// TIA Portal V20 export
FUNCTION "07 T5 EXCENTRIC LEV2" : Void   // FC1718, LAD
TITLE = TRACKING - LEV2
{ S7_Optimized_Access := 'TRUE' }
// stored: AutoNumber false, SetENOAutomatically false
   VAR_TEMP
      "HSK Answer OK" : Bool;
      Trc_OK : Bool;
      Aux_Int : Int;
      Aux_Bool : Bool;
   END_VAR
   VAR_TEMP   // added for the SCL form of the ladder/FBD networks
      _w1 : Bool;
      _w2 : Bool;
      _w3 : Bool;
   END_VAR
BEGIN

REGION Network 1: ============ Manual movement ============
END_REGION

REGION Network 2: pipe trasnfered
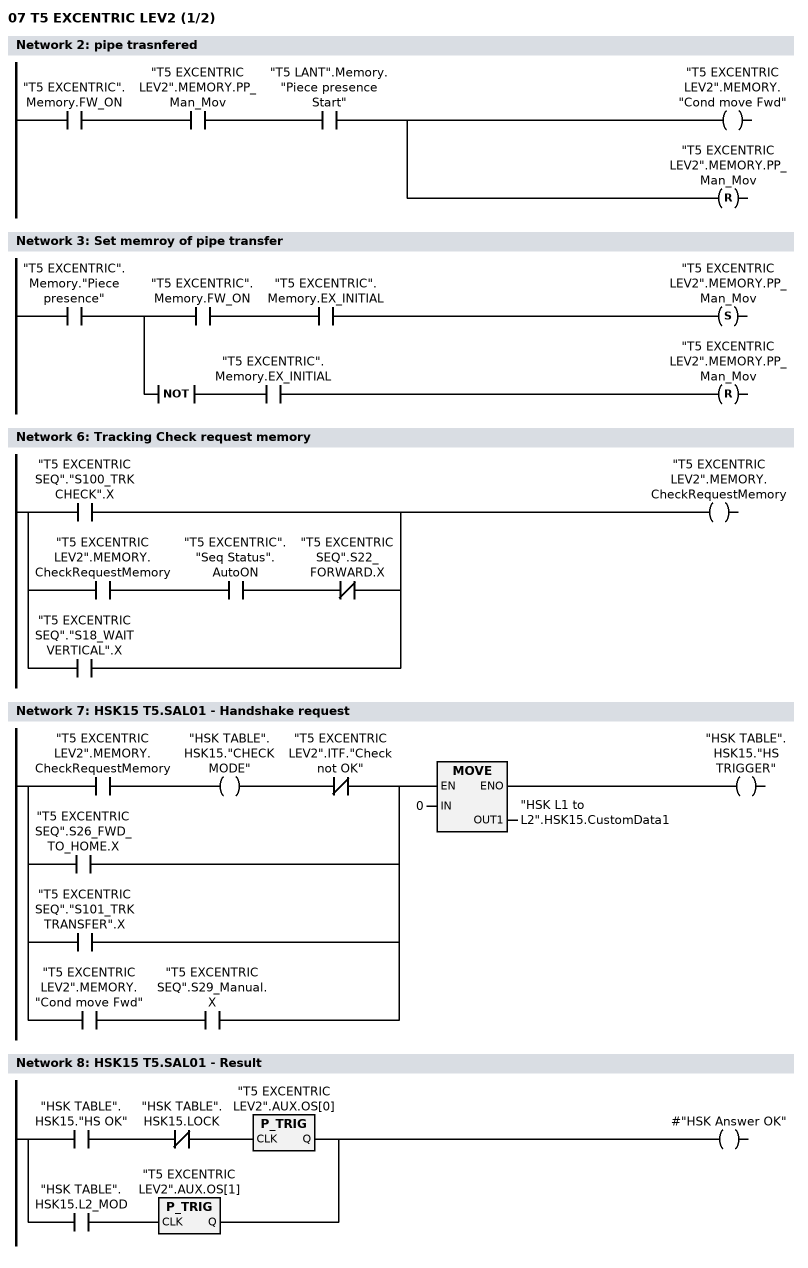
   RUNG wire#powerrail
      Contact( "T5 EXCENTRIC".Memory.FW_ON )
      Contact( "T5 EXCENTRIC LEV2".MEMORY.PP_Man_Mov )
      Contact( "T5 LANT".Memory."Piece presence Start" )
      wire#w1
      Coil( "T5 EXCENTRIC LEV2".MEMORY."Cond move Fwd" )
   END_RUNG
   RUNG wire#w1
      R_Coil( "T5 EXCENTRIC LEV2".MEMORY.PP_Man_Mov )
   END_RUNG
   // the same network as SCL:
   "T5 EXCENTRIC LEV2".MEMORY."Cond move Fwd" := "T5 EXCENTRIC".Memory.FW_ON AND "T5 EXCENTRIC LEV2".MEMORY.PP_Man_Mov AND "T5 LANT".Memory."Piece presence Start";
   IF "T5 EXCENTRIC LEV2".MEMORY."Cond move Fwd" THEN "T5 EXCENTRIC LEV2".MEMORY.PP_Man_Mov := FALSE; END_IF;
END_REGION

REGION Network 3: Set memroy of pipe transfer
   RUNG wire#powerrail
      Contact( "T5 EXCENTRIC".Memory."Piece presence" )
      wire#w1
      Contact( "T5 EXCENTRIC".Memory.FW_ON )
      Contact( "T5 EXCENTRIC".Memory.EX_INITIAL )
      S_Coil( "T5 EXCENTRIC LEV2".MEMORY.PP_Man_Mov )
   END_RUNG
   RUNG wire#w1
      Not()
      Contact( "T5 EXCENTRIC".Memory.EX_INITIAL )
      R_Coil( "T5 EXCENTRIC LEV2".MEMORY.PP_Man_Mov )
   END_RUNG
   // the same network as SCL:
   IF "T5 EXCENTRIC".Memory."Piece presence" AND "T5 EXCENTRIC".Memory.FW_ON AND "T5 EXCENTRIC".Memory.EX_INITIAL THEN
       "T5 EXCENTRIC LEV2".MEMORY.PP_Man_Mov := TRUE;
   END_IF;
   IF NOT "T5 EXCENTRIC".Memory."Piece presence" AND "T5 EXCENTRIC".Memory.EX_INITIAL THEN
       "T5 EXCENTRIC LEV2".MEMORY.PP_Man_Mov := FALSE;
   END_IF;
END_REGION

REGION Network 4: ============ Handshake mamnagement ============
END_REGION

REGION Network 5: ====== HSK15 T5.SAL01 ======
END_REGION

REGION Network 6: Tracking Check request memory
   RUNG wire#powerrail
      Contact( "T5 EXCENTRIC SEQ"."S100_TRK CHECK".X )
      wire#w1
      Coil( "T5 EXCENTRIC LEV2".MEMORY.CheckRequestMemory )
   END_RUNG
   RUNG wire#powerrail
      Contact( "T5 EXCENTRIC LEV2".MEMORY.CheckRequestMemory )
      Contact( "T5 EXCENTRIC"."Seq Status".AutoON )
      I_Contact( "T5 EXCENTRIC SEQ".S22_FORWARD.X )
   END_RUNG wire#w1
   RUNG wire#powerrail
      Contact( "T5 EXCENTRIC SEQ"."S18_WAIT VERTICAL".X )
   END_RUNG wire#w1
   // the same network as SCL:
   "T5 EXCENTRIC LEV2".MEMORY.CheckRequestMemory := "T5 EXCENTRIC SEQ"."S100_TRK CHECK".X OR ("T5 EXCENTRIC LEV2".MEMORY.CheckRequestMemory AND "T5 EXCENTRIC"."Seq Status".AutoON AND NOT "T5 EXCENTRIC SEQ".S22_FORWARD.X) OR "T5 EXCENTRIC SEQ"."S18_WAIT VERTICAL".X;
END_REGION

REGION Network 7: HSK15 T5.SAL01 - Handshake request
   RUNG wire#powerrail
      Contact( "T5 EXCENTRIC LEV2".MEMORY.CheckRequestMemory )
      Coil( "HSK TABLE".HSK15."CHECK MODE" )
      I_Contact( "T5 EXCENTRIC LEV2".ITF."Check not OK" )
      wire#w1
      Move(in := 0, out1 => "HSK L1 to L2".HSK15.CustomData1)
      Coil( "HSK TABLE".HSK15."HS TRIGGER" )
   END_RUNG
   RUNG wire#powerrail
      Contact( "T5 EXCENTRIC SEQ".S26_FWD_TO_HOME.X )
   END_RUNG wire#w1
   RUNG wire#powerrail
      Contact( "T5 EXCENTRIC SEQ"."S101_TRK TRANSFER".X )
   END_RUNG wire#w1
   RUNG wire#powerrail
      Contact( "T5 EXCENTRIC LEV2".MEMORY."Cond move Fwd" )
      Contact( "T5 EXCENTRIC SEQ".S29_Manual.X )
   END_RUNG wire#w1
   // the same network as SCL:
   "HSK TABLE".HSK15."CHECK MODE" := "T5 EXCENTRIC LEV2".MEMORY.CheckRequestMemory;
   #_w1 := ("T5 EXCENTRIC LEV2".MEMORY.CheckRequestMemory AND NOT "T5 EXCENTRIC LEV2".ITF."Check not OK") OR "T5 EXCENTRIC SEQ".S26_FWD_TO_HOME.X OR "T5 EXCENTRIC SEQ"."S101_TRK TRANSFER".X OR ("T5 EXCENTRIC LEV2".MEMORY."Cond move Fwd" AND "T5 EXCENTRIC SEQ".S29_Manual.X);
   IF #_w1 THEN "HSK L1 to L2".HSK15.CustomData1 := 0; END_IF;
   "HSK TABLE".HSK15."HS TRIGGER" := #_w1;
END_REGION

REGION Network 8: HSK15 T5.SAL01 - Result
   RUNG wire#powerrail
      Contact( "HSK TABLE".HSK15."HS OK" )
      I_Contact( "HSK TABLE".HSK15.LOCK )
      P_Trig( "T5 EXCENTRIC LEV2".AUX.OS[0] )
      wire#w1
      Coil( #"HSK Answer OK" )
   END_RUNG
   RUNG wire#powerrail
      Contact( "HSK TABLE".HSK15.L2_MOD )
      P_Trig( "T5 EXCENTRIC LEV2".AUX.OS[1] )
   END_RUNG wire#w1
   // the same network as SCL:
   #_w1 := "HSK TABLE".HSK15."HS OK" AND NOT "HSK TABLE".HSK15.LOCK;
   #_w2 := #_w1 AND NOT "T5 EXCENTRIC LEV2".AUX.OS[0];   // rising edge
   "T5 EXCENTRIC LEV2".AUX.OS[0] := #_w1;
   #_w3 := "HSK TABLE".HSK15.L2_MOD AND NOT "T5 EXCENTRIC LEV2".AUX.OS[1];   // rising edge
   "T5 EXCENTRIC LEV2".AUX.OS[1] := "HSK TABLE".HSK15.L2_MOD;
   #"HSK Answer OK" := #_w2 OR #_w3;
END_REGION

REGION Network 9: Check OK / not OK
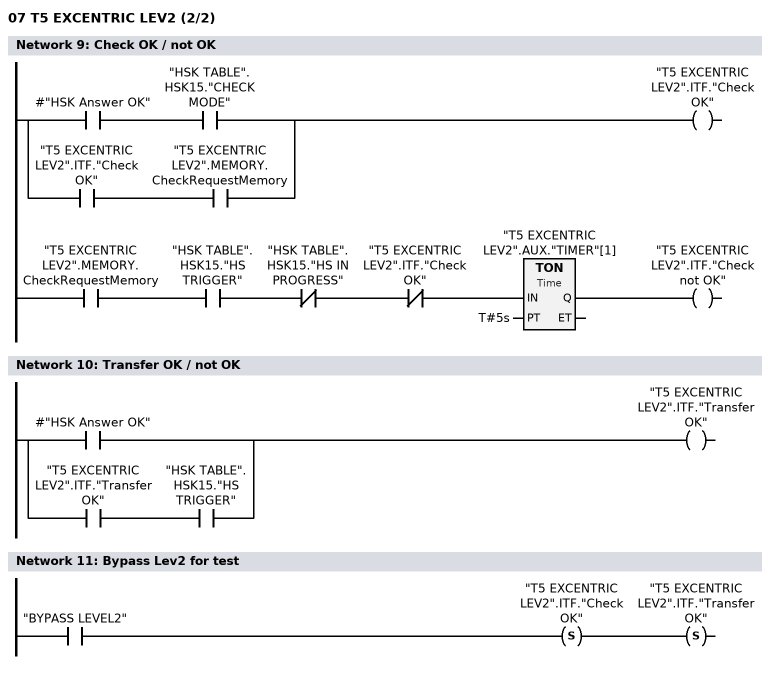
   RUNG wire#powerrail
      Contact( #"HSK Answer OK" )
      Contact( "HSK TABLE".HSK15."CHECK MODE" )
      wire#w1
      Coil( "T5 EXCENTRIC LEV2".ITF."Check OK" )
   END_RUNG
   RUNG wire#powerrail
      Contact( "T5 EXCENTRIC LEV2".ITF."Check OK" )
      Contact( "T5 EXCENTRIC LEV2".MEMORY.CheckRequestMemory )
   END_RUNG wire#w1
   RUNG wire#powerrail
      Contact( "T5 EXCENTRIC LEV2".MEMORY.CheckRequestMemory )
      Contact( "HSK TABLE".HSK15."HS TRIGGER" )
      I_Contact( "HSK TABLE".HSK15."HS IN PROGRESS" )
      I_Contact( "T5 EXCENTRIC LEV2".ITF."Check OK" )
      { S7_Templates := "time_type := Time" } "T5 EXCENTRIC LEV2".AUX."TIMER"[1].TON(pt := T#5s, et =>)
      Coil( "T5 EXCENTRIC LEV2".ITF."Check not OK" )
   END_RUNG
   // the same network as SCL:
   "T5 EXCENTRIC LEV2".ITF."Check OK" := (#"HSK Answer OK" AND "HSK TABLE".HSK15."CHECK MODE") OR ("T5 EXCENTRIC LEV2".ITF."Check OK" AND "T5 EXCENTRIC LEV2".MEMORY.CheckRequestMemory);
   "T5 EXCENTRIC LEV2".AUX."TIMER"[1].TON(IN := "T5 EXCENTRIC LEV2".MEMORY.CheckRequestMemory AND "HSK TABLE".HSK15."HS TRIGGER" AND NOT "HSK TABLE".HSK15."HS IN PROGRESS" AND NOT "T5 EXCENTRIC LEV2".ITF."Check OK",
                           PT := T#5s);
   "T5 EXCENTRIC LEV2".ITF."Check not OK" := "T5 EXCENTRIC LEV2".AUX."TIMER"[1].Q;
END_REGION

REGION Network 10: Transfer OK / not OK
   RUNG wire#powerrail
      Contact( #"HSK Answer OK" )
      wire#w1
      Coil( "T5 EXCENTRIC LEV2".ITF."Transfer OK" )
   END_RUNG
   RUNG wire#powerrail
      Contact( "T5 EXCENTRIC LEV2".ITF."Transfer OK" )
      Contact( "HSK TABLE".HSK15."HS TRIGGER" )
   END_RUNG wire#w1
   // the same network as SCL:
   "T5 EXCENTRIC LEV2".ITF."Transfer OK" := #"HSK Answer OK" OR ("T5 EXCENTRIC LEV2".ITF."Transfer OK" AND "HSK TABLE".HSK15."HS TRIGGER");
END_REGION

REGION Network 11: Bypass Lev2 for test
   RUNG wire#powerrail
      Contact( "BYPASS LEVEL2" )
      S_Coil( "T5 EXCENTRIC LEV2".ITF."Check OK" )
      S_Coil( "T5 EXCENTRIC LEV2".ITF."Transfer OK" )
   END_RUNG
   // the same network as SCL:
   IF "BYPASS LEVEL2" THEN
       "T5 EXCENTRIC LEV2".ITF."Check OK" := TRUE;
       "T5 EXCENTRIC LEV2".ITF."Transfer OK" := TRUE;
   END_IF;
END_REGION
END_FUNCTION
